(* IEC 61131-3 sources: ConveyorControl-with-PLC/4E_Gruppe1_Graf_Projekt1/Class/Abschluss, 1 file *)

(* ---- Abschluss.st ---- *)
(*!
<Class
	Name               = "Abschluss"
	Revision           = "0.0"
	RealtimeTask       = "false"
	CyclicTask         = "true"
	DefCyclictime      = "10 ms"
	BackgroundTask     = "false"
	Sigmatek           = "false"
	OSInterface        = "false"
	HighPriority       = "false"
	Automatic          = "false"
	UpdateMode         = "Prescan"
	SharedCommandTable = "true"
	Objectsize         = "(398,120)">
	<Channels>
		<Server Name="Alarm" Visualized="true" Initialize="false" WriteProtected="false" Retentive="false"/>
		<Server Name="auto" Visualized="true" Initialize="false" WriteProtected="false" Retentive="false"/>
		<Server Name="auto_spd" Visualized="true" Initialize="true" DefValue="500" WriteProtected="false" Retentive="false"/>
		<Server Name="ClassSvr" Visualized="false" Initialize="false" WriteProtected="true" Retentive="false"/>
		<Server Name="hand" Visualized="true" Initialize="false" WriteProtected="false" Retentive="false"/>
		<Server Name="input_S1" Visualized="true" Initialize="false" WriteProtected="false" Retentive="false"/>
		<Server Name="input_S2" Visualized="true" Initialize="false" WriteProtected="false" Retentive="false"/>
		<Server Name="input_S3" Visualized="true" Initialize="false" WriteProtected="false" Retentive="false"/>
		<Server Name="spd" Visualized="false" Initialize="false" WriteProtected="false" Retentive="false"/>
		<Server Name="status" Visualized="false" Initialize="false" WriteProtected="false" Retentive="false"/>
		<Server Name="stop" Visualized="true" Initialize="false" WriteProtected="false" Retentive="false"/>
		<Client Name="MTR_enable" Required="true" Internal="false"/>
		<Client Name="MTR_speed" Required="true" Internal="false"/>
	</Channels>
</Class>
*)
Abschluss : CLASS
	TYPE
	  state_type :  //! <Type Public="true" Name="state_type"/>
	  (
	    waitForInput:=0,
	    auto_mtr_on:=1,
	    auto_mtr_fill:=2,
	    hand_active:=3,
	    err
	  )$UDINT;
	END_TYPE
  //Servers:
	ClassSvr 	: SvrChCmd_DINT;
	status 	: SvrCh_state_type_PTofCls_Abschluss;
	auto 	: SvrCh_DINT;
	spd 	: SvrCh_DINT;
	hand 	: SvrCh_DINT;
	input_S1 	: SvrCh_DINT;
	input_S2 	: SvrCh_DINT;
	input_S3 	: SvrCh_DINT;
	stop 	: SvrCh_DINT;
	Alarm 	: SvrCh_DINT;
	auto_spd 	: SvrCh_DINT;
  //Clients:
	MTR_speed 	: CltCh_DINT;
	MTR_enable 	: CltCh_DINT;
  //Variables:
  //Functions:

	FUNCTION VIRTUAL GLOBAL CyWork
		VAR_INPUT
			EAX 	: UDINT;
		END_VAR
		VAR_OUTPUT
			state (EAX) 	: UDINT;
		END_VAR;
  //Tables:
	FUNCTION @STD
		VAR_OUTPUT
			ret_code	: CONFSTATES;
		END_VAR;
	FUNCTION GLOBAL TAB @CT_;
END_CLASS;

FUNCTION VIRTUAL GLOBAL Abschluss::CyWork
	VAR_INPUT
		EAX 	: UDINT;
	END_VAR
	VAR_OUTPUT
		state (EAX) 	: UDINT;
	END_VAR

    if input_S3 = 1 or stop = 1 then
      Alarm:=1;
      stop:=1;
      MTR_enable := 0;
      status := err;
      else
        Alarm:=0;
    end_if;

    if hand = 1 then
      status := hand_active;
    else
      if auto = 1 then
        status := auto_mtr_on;
        else if status = hand_active or stop = 1 then
              status := waitForInput;
             end_if;

      end_if;
    end_if;

  case status of
    err:

    waitForInput:
      Alarm := 2;
      if stop = 1 then
        Alarm := 1;
      end_if;

      spd := 0;
      MTR_enable := 0;

    auto_mtr_on:
      MTR_enable := 1;
      spd := auto_spd;
      if input_S1 = 1 then
        status := auto_mtr_fill;
      end_if;

    auto_mtr_fill:
      MTR_enable := 0;
      spd := 0;
      if input_S2 = 1 then
        status := auto_mtr_on;
      end_if;

    hand_active:
      MTR_enable := 1;
      spd := auto_spd*2;

  end_case;

  MTR_speed.Write (spd);
  MTR_enable.Write (MTR_enable);

	state := READY;

END_FUNCTION
